DATA_BLOCK "SIRENE_DB"
{ S7_Optimized_Access := 'TRUE' }
VERSION : 0.1
NON_RETAIN
"SIRENE"

BEGIN

END_DATA_BLOCK

